{attribute 'strict'}
TYPE E_FcqRobotActions :
(
	FCQ_ROBOT_ACTION_PICK					:= 60,
	FCQ_ROBOT_ACTION_PLACE					:= 61,
	FCQ_ROBOT_ACTION_GO_TO_TRAYFEEDER		:= 62,
	FCQ_ROBOT_ACTION_GO_FIXTURE_ONE_PLACE	:= 63,
	FCQ_ROBOT_ACTION_GO_FIXTURE_ONE_PICK	:= 64,
	FCQ_ROBOT_ACTION_GO_FIXTURE_TWO_PLACE	:= 65,
	FCQ_ROBOT_ACTION_GO_FIXTURE_TWO_PICK	:= 66,
	FCQ_ROBOT_ACTION_GO_FIXTURE_THREE_PLACE	:= 67,
	FCQ_ROBOT_ACTION_GO_FIXTURE_THREE_PICK	:= 68,
	FCQ_ROBOT_ACTION_GO_FIXTURE_FOUR_PLACE	:= 69,
	FCQ_ROBOT_ACTION_GO_FIXTURE_FOUR_PICK	:= 70,
	FCQ_ROBOT_ACTION_GO_TO_ROTARY_TABLE		:= 71,
	FCQ_ROBOT_ACTION_GO_SAFE_POSITION		:= 72,
	FCQ_ROBOT_ACTION_GO_INPUT_PRODUCT		:= 73,
	FCQ_ROBOT_ACTION_GO_OUTPUT_PRODUCT		:= 74,
	FCQ_ROBOT_ACTION_GO_TO_GS_HIGH_1		:= 75,
	FCQ_ROBOT_ACTION_GO_TO_GS_HIGH_2		:= 76,
	FCQ_ROBOT_ACTION_GO_TO_GS_HIGH_3		:= 77,
	FCQ_ROBOT_ACTION_GO_TO_GS_HIGH_4		:= 78,
	FCQ_ROBOT_ACTION_GO_TO_GS_LOW_1			:= 79,
	FCQ_ROBOT_ACTION_GO_TO_GS_LOW_2			:= 80,
	FCQ_ROBOT_ACTION_GO_TO_GS_LOW_3			:= 81,
	FCQ_ROBOT_ACTION_GO_TO_GS_LOW_4			:= 82,
	FCQ_ROBOT_ACTION_PLACE_RNR				:= 83,
	FCQ_ROBOT_ACTION_PICK_RNR				:= 84,
	FCQ_ROBOT_ACTION_GO_INPUT_RNR			:= 85
)UINT;
END_TYPE

(* stored: Version 1.1.0.1, ProductVersion 3.1.4024.9
   DUT E_FcqRobotActions: Id {1cc4a311-0c01-4418-93a2-204d601852a7} *)
